// TwinCAT 3 PLC project AA_Planta_2324_MN
// ProgramVersion: 3.1.4024.0
// libraries:
//   Tc2_Standard, * (Beckhoff Automation GmbH)
//   Tc2_System, * (Beckhoff Automation GmbH)
//   Tc3_Module, * (Beckhoff Automation GmbH)
// project tree:
//   DUTs/ COLOR.TcDUT
//   DUTs/DefinicionCases/ CALMACENAMIENTO.TcDUT, CINTA.TcDUT, CPICKANDPLACE.TcDUT, CPOSITIONERLEFTBAR.TcDUT, CONDICIONESPARO.TcDUT, CRETIRADA.TcDUT, CTURNTABLE.TcDUT, STOPBLADE.TcDUT
//   DUTs/Objetos/ BeltConveyor.TcDUT, PickandPlace.TcDUT, PositioningLeftBar.TcDUT, Pusher.TcDUT, RollerConveyor.TcDUT, Selector.TcDUT, StrackerCraneRack.TcDUT, Turntable.TcDUT
//   GVLs/ GVL_General.TcGVL, GVL_ProcesoPallet.TcGVL, GVL_Sorting.TcGVL, GVL_StackBox.TcGVL, GVL_Almacen.TcGVL
//   / PlcTask.TcTTO
//   POUs/0_ControlEncendido/ PRG_FinDeCiclo.TcPOU, PRG_OnFabrica.TcPOU, PRG_SetaEmergencia.TcPOU, PRG_StopBladePyP.TcPOU
//   POUs/3_ProcesoPalet/ PRG_Cintas.TcPOU, PRG_Turntable.TcPOU
//   POUs/4_Almacen/ DINT_TO_COLOR.TcPOU, PRG_Almacen.TcPOU, PRG_PanelDeControl.TcPOU, PRG_RetiradaAlmacen.TcPOU
//   POUs/6_Contadores/ POU_Contadores.TcPOU
//   POUs/ MAIN.TcPOU
//   POUs/1_ProcesoEntrada/ FB_Pusher.TcPOU, PRG_ProcesoEntrada.TcPOU
//   POUs/2_ProcesoGuardado/ FB_Cinta.TcPOU, FB_PickAndPlace.TcPOU, FB_Positioner.TcPOU, FB_StopBlade.TcPOU, PRG_Parada.TcPOU, PRG_PickAndPlace.TcPOU, PRG_Positioner.TcPOU
// real-time tasks:
//   TASK PlcTask: cycle T#10ms, priority 20, ADS port 350
//   TASK PlcTask1: cycle T#10ms, priority 21, ADS port 351

CONFIGURATION AA_Planta_2324_MN
    RESOURCE PLC ON TwinCAT3
        TASK PlcTask(INTERVAL := T#10ms, PRIORITY := 21);
        PROGRAM MAIN WITH PlcTask : MAIN;
    END_RESOURCE
END_CONFIGURATION

// ---- DUTs/COLOR.TcDUT
{attribute 'strict'}
TYPE COLOR :
(
	AZUL := 2,
	VERDE := 5,
	METAL := 8,
	VACIO := 0
);
END_TYPE

// ---- DUTs/DefinicionCases/CALMACENAMIENTO.TcDUT
{attribute 'strict'}
TYPE CALMACENAMIENTO :
(
	CALMACEN_ESPERA,
	CALMACEN_MONTARPALLET,
	CALMACEN_BUSQUEDA,
	CALMACEN_GUARDADO,
	CALMACEN_LLENO,
	CALMACEN_ORIGEN
	
);
END_TYPE

// ---- DUTs/DefinicionCases/CINTA.TcDUT
{attribute 'strict'}
TYPE CINTA :
(
	CINTA_ACTIVADO,
	CINTA_REPOSO
);
END_TYPE

// ---- DUTs/DefinicionCases/CPICKANDPLACE.TcDUT
{attribute 'strict'}
TYPE CPICKANDPLACE :
(
	PICKANDPLACE_ESPERA,
	PICKANDPLACE_DETECCION,
	PICKANDPLACE_AGARRE,
	PICKANDPLACE_GIRO,
	PICKANDPLACE_COLOCACION,
	PICKANDPLACE_DESCENSO,
	PICKANDPLACE_LLENADO,
	PICKANDPLACE_ORIGEN
);
END_TYPE

// ---- DUTs/DefinicionCases/CPOSITIONERLEFTBAR.TcDUT
{attribute 'strict'}
TYPE CPOSITIONERLEFTBAR :
(
	CPOSITIONERLEFTBAR_ESPERA,
	CPOSITIONERLEFTBAR_AGARRE,
	CPOSITIONERLEFTBAR_PROCESADO,
	CPOSITIONERLEFTBAR_RESET,
	CPOSITIONERLEFTBAR_PASO
	
	
);
END_TYPE

// ---- DUTs/DefinicionCases/CONDICIONESPARO.TcDUT
{attribute 'strict'}
TYPE CONDICIONESPARO :
(
	CONDICIONESPARO_ESPERA,
	CONDICIONESPARO_SELECCION,
	CONDICIONESPARO_FINPROCESO,
	CONDICIONESPARO_ALMACEN,
	CONDICIONESPARO_SELECTOR,
	CONDICIONESPARO_GUARDADO,
	CONDICIONESPARO_CINTAINICIAL
);
END_TYPE

// ---- DUTs/DefinicionCases/CRETIRADA.TcDUT
{attribute 'strict'}
TYPE CRETIRADA :
(
	CRETIRADA_ESPERA,
	CRETIRADA_BUSQUEDA,
	CRETIRADA_RECOGIDA,
	CRETIRADA_TRANSPORTE,
	CRETIRADA_COLOCACION,
	CRETIRADA_PARTIDA
);
END_TYPE

// ---- DUTs/DefinicionCases/CTURNTABLE.TcDUT
{attribute 'strict'}
TYPE CTURNTABLE :
(
	CTURNTABLE_ESPERA,
	CTURNTABLE_FILTROPRIORIDAD,
	
	CTURNTABLE_ENTRADAVERDE,
	CTURNTABLE_CARGAVERDE,
	CTURNTABLE_DESCARGAVERDE,
	
	CTURNTABLE_ENTRADAAZUL,
	CTURNTABLE_CARGAAZUL,
	CTURNTABLE_DESCARGAAZUL,
	
	CTURNTABLE_ENTRADAMETAL,
	CTURNTABLE_CARGAMETAL,
	CTURNTABLE_DESCARGAMETAL,
	
	CTURNTABLE_COLOCACION,
	CTURNTABLE_SALIDA
);
END_TYPE

// ---- DUTs/DefinicionCases/STOPBLADE.TcDUT
{attribute 'strict'}
TYPE STOPBLADE :
(
	STOPBLADE_REPOSO,
	STOPBLADE_ACTIVADO
);
END_TYPE

// ---- DUTs/Objetos/BeltConveyor.TcDUT
{attribute 'OPC.UA.DA' := '1'}
TYPE BeltConveyor :
STRUCT
	
	(* Cintas comunes correspondientes al proceso de Sorting, ordenadas por aparición*)
	bSortingCintaInicial		: BOOL;
	bSortingCintaEntrada		: BOOL;
	bSortingCintaDistribucion	: BOOL;
	
	(* Cintas PARA PIEZAS AZULES, ordenadas por aparición*)
	bCintaAzul1 	: BOOL;
	bCintaAzul2		: BOOL;
	
	(* Cintas PARA PIEZAS VERDES, ordenadas por aparición*)
	bCintaVerde1 	: BOOL;
	bCintaVerde2	: BOOL;

	(* Cintas PARA PIEZAS METAL, ordenadas por aparición*)
	bCintaMetal1 	: BOOL;
	bCintaMetal2	: BOOL;
	
END_STRUCT
END_TYPE

// ---- DUTs/Objetos/PickandPlace.TcDUT
{attribute 'OPC.UA.DA' := '1'}
TYPE PickandPlace :
STRUCT
	
	(* Outputs del Pick and Place *)
 	bMovementZ 	: BOOL;
 	bMovementX 	: BOOL;
	bRotateCW 	: BOOL;
	bRotateCCW 	: BOOL;
	bGripperCW 	: BOOL;
	bGripperCCW : BOOL;
	bGrab 		: BOOL;
	
	(* Inputs del Pick and Place *)
	bMovingX 			: BOOL;
	bMovingZ 			: BOOL;
	bRotating 			: BOOL;
	bGripperRotating	: BOOL;
	bDetected 			: BOOL;

END_STRUCT
END_TYPE

// ---- DUTs/Objetos/PositioningLeftBar.TcDUT
{attribute 'OPC.UA.DA' := '1'}
TYPE PositioningLeftBar :
STRUCT
	
	(* Outputs del Positioning Left Bar *)
	bClamp : BOOL;
	bRaise : BOOL;
	
	(* Inputs del Positioning Left Bar *)
	bClamped : BOOL;
	bLimit	 : BOOL;
	
END_STRUCT
END_TYPE

// ---- DUTs/Objetos/Pusher.TcDUT
{attribute 'OPC.UA.DA' := '1'}
TYPE Pusher :
STRUCT
	Pusher: BOOL;
	PusherFrontLimit: BOOL;
	PusherBackLimit: BOOL;
END_STRUCT
END_TYPE

// ---- DUTs/Objetos/RollerConveyor.TcDUT
{attribute 'OPC.UA.DA' := '1'}
TYPE RollerConveyor :
STRUCT
	
	(* ROLL PARA PIEZAS AZULES, ordenadas por aparición*)
	bRollerAzul1 		 : BOOL;
	bCurvedRollerAzul1 	 : BOOL;
	
	(* ROLL PARA PIEZAS VERDES, ordenadas por aparición*)
	bRollerVerde1 		 : BOOL;
	
	(* ROLL PARA PIEZAS METAL, ordenadas por aparición*)
	bRollerMetal1 		 : BOOL;
	bCurvedRollerMetal1  : BOOL;
	
	(* ROLL ALMACEN, ordenadas por aparición*)
	bRollerAlmacen1		 : BOOL;
	bCurvedRollerAlmacen : BOOL;
	bRollerAlmacen2		 : BOOL;
	
	(* ROLLER SALIDA ALMACEN, ordenadas por aparición *)
	
	bRollerAlmacen3 : BOOL;
	bRollerAlmacen4 : BOOL;
	
END_STRUCT
END_TYPE

// ---- DUTs/Objetos/Selector.TcDUT
{attribute 'OPC.UA.DA' := '1'}
TYPE Selector :
STRUCT
	StateAzul : BOOL;
	StateMetal : BOOL;
END_STRUCT
END_TYPE

// ---- DUTs/Objetos/StrackerCraneRack.TcDUT
{attribute 'OPC.UA.DA' := '1'}
TYPE StrackerCraneRack :
STRUCT
	
	(* Outputs del Almacen *)
	TargetPosition: INT;
	Left:BOOL;
	Right:BOOL;
	Lift:BOOL;
	
	(* Inputs del Almacen *)
	MovingX:BOOL;
	MovingZ:BOOL;
	LeftLimit:BOOL;
	MiddleLimit:BOOL;
	RightLimit:BOOL;
	
END_STRUCT
END_TYPE

// ---- DUTs/Objetos/Turntable.TcDUT
{attribute 'OPC.UA.DA' := '1'}
TYPE Turntable :
STRUCT
	
	(* Outputs de la Turntable *)
	RollPositivo : BOOL;
	RollNegativo : BOOL;
	Turn		 : BOOL;
	
	(* Inputs de la Turntable *)
	FrontLimit	 : BOOL;
	BackLimit	 : BOOL;
	Limit0		 : BOOL;
	Limit90		 : BOOL;
	
END_STRUCT
END_TYPE

// ---- GVLs/GVL_General.TcGVL
{attribute 'qualified_only'}
VAR_GLOBAL
	{attribute 'OPC.UA.DA' := '1'}
	bMarcha : BOOL;
	{attribute 'OPC.UA.DA' := '1'}
	bParo : BOOL;
	{attribute 'OPC.UA.DA' := '1'}
	bSetaEmergencia : BOOL;
	
	{attribute 'OPC.UA.DA.StructuredType' := '1'}
	sBeltConveyor: BeltConveyor;
	
	{attribute 'OPC.UA.DA' := '1'}
	bStopBlade1 : BOOL;	
	
END_VAR

// ---- GVLs/GVL_ProcesoPallet.TcGVL
{attribute 'qualified_only'}
VAR_GLOBAL	
	
	{attribute 'OPC.UA.DA.StructuredType' := '1'}
	sTurnTable: Turntable;
	{attribute 'OPC.UA.DA.StructuredType' := '1'}
	sRollerConveyor: RollerConveyor;
	
	{attribute 'OPC.UA.DA' := '1'}
	bDiffuseSensorPaletA	:BOOL;
	{attribute 'OPC.UA.DA' := '1'}
	bDiffuseSensorPaletV	:BOOL;
	{attribute 'OPC.UA.DA' := '1'}
	bDiffuseSensorPaletM	:BOOL;
	{attribute 'OPC.UA.DA' := '1'}	
	bDiffuseSensorSalida		:BOOL;
	
	{attribute 'OPC.UA.DA' := '1'}
	iLightArrayEmitterA		:BOOL;
	{attribute 'OPC.UA.DA' := '1'}
	iLightArrayEmitterV		:BOOL;
	{attribute 'OPC.UA.DA' := '1'}
	iLightArrayEmitterM		:BOOL; 
	
END_VAR

// ---- GVLs/GVL_Sorting.TcGVL
{attribute 'qualified_only'}
VAR_GLOBAL

	(* Variables correspondientes al proceso de sorting de las piezas AZULES *)
	{attribute 'OPC.UA.DA' := '1'}
	bVisionSensorA	: BOOL;
	{attribute 'OPC.UA.DA.StructuredType' := '1'}
	sPusherA: Pusher;
	{attribute 'OPC.UA.DA' := '1'}
	bDiffuseSensorA: BOOL;
	
	(* Variables correspondientes al proceso de sorting de las piezas VERDES *)
	{attribute 'OPC.UA.DA.StructuredType' := '1'}
	sPusherV: Pusher;
	{attribute 'OPC.UA.DA' := '1'}
	bVisionSensorV	: BOOL;	
	{attribute 'OPC.UA.DA' := '1'}
	bDiffuseSensorV: BOOL;
	
	(* Variables correspondientes al proceso de sorting de las piezas METÁLICAS *)
	{attribute 'OPC.UA.DA.StructuredType' := '1'}
	sPusherM: Pusher;
	{attribute 'OPC.UA.DA' := '1'}
	bVisionSensorM	: BOOL;
	{attribute 'OPC.UA.DA' := '1'}
	bDiffuseSensorM: BOOL;
	
END_VAR

// ---- GVLs/GVL_StackBox.TcGVL
{attribute 'qualified_only'}
VAR_GLOBAL
	
	(* Variables correspondientes a la Línea Azul*)
	
	{attribute 'OPC.UA.DA.StructuredType' := '1'}
	sPickAndPlaceA	: PickAndPlace;
	{attribute 'OPC.UA.DA.StructuredType' := '1'}
	sPosLeftBarA	: PositioningLeftBar;
	{attribute 'OPC.UA.DA' := '1'}
	bStopBladeA1: BOOL;
	{attribute 'OPC.UA.DA' := '1'}
	bStopBladeA2: BOOL := TRUE;
	
	{attribute 'OPC.UA.DA' := '1'}
	bRReflectiveSensorA1 	: BOOL	:= TRUE;
	{attribute 'OPC.UA.DA' := '1'}
	bRReflectiveSensorA2 	: BOOL	:= TRUE;
	{attribute 'OPC.UA.DA' := '1'}
	bRReflectiveSensorA3	: BOOL	:= TRUE;
	{attribute 'OPC.UA.DA' := '1'}
	bDiffuseSensorPyPA		: BOOL	:= FALSE;
	

	
	(* Variables correspondientes a la Línea Verde*)
	
	{attribute 'OPC.UA.DA.StructuredType' := '1'}
	sPickAndPlaceV	: PickAndPlace;
	{attribute 'OPC.UA.DA.StructuredType' := '1'}
	sPosLeftBarV	: PositioningLeftBar;
	{attribute 'OPC.UA.DA' := '1'}
	bStopBladeV1: BOOL;
	{attribute 'OPC.UA.DA' := '1'}
	bStopBladeV2: BOOL := TRUE;
	
	
	{attribute 'OPC.UA.DA' := '1'}
	bRReflectiveSensorV1 : BOOL		:= TRUE;
	{attribute 'OPC.UA.DA' := '1'}
	bRReflectiveSensorV2 : BOOL		:= TRUE;
	{attribute 'OPC.UA.DA' := '1'}	
	bRReflectiveSensorV3 : BOOL		:= TRUE;
	{attribute 'OPC.UA.DA' := '1'}	
	bDiffuseSensorPyPV	 : BOOL		:= FALSE;
	
	
	
	(* Variables correspondientes a la Línea Metal*)
	
	{attribute 'OPC.UA.DA.StructuredType' := '1'}
	sPickAndPlaceM	: PickAndPlace;
	{attribute 'OPC.UA.DA.StructuredType' := '1'}
	sPosLeftBarM	: PositioningLeftBar;
	{attribute 'OPC.UA.DA' := '1'}
	bStopBladeM1: BOOL;
	{attribute 'OPC.UA.DA' := '1'}
	bStopBladeM2: BOOL := TRUE;
	
	{attribute 'OPC.UA.DA' := '1'}
	bRReflectiveSensorM1 : BOOL		:= TRUE;
	{attribute 'OPC.UA.DA' := '1'}
	bRReflectiveSensorM2 : BOOL		:= TRUE;
	{attribute 'OPC.UA.DA' := '1'}
	bRReflectiveSensorM3 : BOOL		:= TRUE;
	{attribute 'OPC.UA.DA' := '1'}
	bDiffuseSensorPyPM	 : BOOL		:= FALSE;

END_VAR

// ---- GVLs/GVL_Almacen.TcGVL
{attribute 'qualified_only'}
VAR_GLOBAL
	
	(* Sensores y actuadores asociados al ciclo del Almacén*)
	
	{attribute 'OPC.UA.DA.StructuredType' := '1'}
	sStackCraneRack: StrackerCraneRack;
	
	{attribute 'OPC.UA.DA' := '1'}
	bDifusseSensorAlmacen:BOOL;
	{attribute 'OPC.UA.DA' := '1'}
	iVisionSensorAlmacen: DINT;
	{attribute 'OPC.UA.DA' := '1'}
	bRRflexSensorAlmacen:BOOL;
	
	{attribute 'OPC.UA.DA' := '1'}
	bLoadingConveyor:BOOL;
	
	(* Almacenamiento de datos de las diferentes posiciones (no es necesario que sea una GVL) *)
	aAlmacen: ARRAY[1..54] OF COLOR  :=[54(0)];
	

	(* Memoria del color solicitado (no es necesario que sea una GVL) *)
	iSolicitudColor : INT;
	
	(* Botones de activación, paro y seta y elementos asociados al panel del Almacén *)
	
	{attribute 'OPC.UA.DA' := '1'}
	Sacar: BOOL;
	{attribute 'OPC.UA.DA' := '1'}
	bReset: BOOL;
	{attribute 'OPC.UA.DA' := '1'}
	bSetaEmergencia: BOOL;
	
	{attribute 'OPC.UA.DA.StructuredType' := '1'}
	sSelector : Selector;
	
	{attribute 'OPC.UA.DA' := '1'}
	iDisplay : INT;
	{attribute 'OPC.UA.DA' := '1'}
	LedAzul: BOOL;
	{attribute 'OPC.UA.DA' := '1'}
	LedVerde: BOOL;
	{attribute 'OPC.UA.DA' := '1'}
	LedMetal: BOOL;
	
END_VAR

// ---- POUs/MAIN.TcPOU
PROGRAM MAIN
VAR
	bON: BOOL; 
END_VAR

(*
  	  ESCOLA POLITÉCNICA DE ENXEÑARÍA DE FERROL			
			  UNIVERSIDADE DA CORUÑA 						
			
Máster Universitario en Informática Industrial y Robótica   
  	Automatización Avanzada - Curso 2023-2024			

					Profesorado: 						
 	Antonio J. Díaz Longueira - Míriam Timiraos Díaz 		

 		    	Código realizado por:
	Marta María Álvarez Crespo - Noelia Pita López  		
*)



(* PRGs siempre activos, necesarios para el correcto control de la fábrica *)
PRG_StopBladePyP();
POU_Contadores();


(* Cuando se pulsa el botón verde, se activa la fábrica y solo se detendrá en caso de que se pulse el botón de paro o la seta de emergencia.
En el caso del botón de paro, desactivará el valor de bON de forma que se llame a un POU diferente a los llamados en este MAIN, donde el proceso
se detiene progresivamente *)

IF GVL_General.bMarcha THEN
	bON := TRUE;
END_IF

IF NOT GVL_General.bParo THEN
	bON := FALSE;
END_IF

IF NOT bON THEN
	PRG_FinDeCiclo();
END_IF


IF bON AND GVL_General.bSetaEmergencia THEN
	
	PRG_OnFabrica();
	PRG_ProcesoEntrada();
	PRG_PickAndPlace();
	PRG_Positioner();
	PRG_Parada();
	PRG_Turntable();
	PRG_Almacen();
	PRG_Cintas();
	PRG_PaneldeControl();
	
	IF GVL_Almacen.bSetaEmergencia THEN
		PRG_RetiradaAlmacen();
	END_IF
	
END_IF

IF NOT GVL_General.bSetaEmergencia THEN
	PRG_SetaEmergencia();
END_IF





























































(*
		♡ 
    /\_____/\
   /  o   o  \						
  ( ==  ^  == )		
   )         (		   __     miau
 (             )______/  |		miau 
(__(__)___(__)__)_______/	 

*)

END_PROGRAM

// ---- POUs/0_ControlEncendido/PRG_StopBladePyP.TcPOU
PROGRAM PRG_StopBladePyP
VAR
END_VAR

GVL_StackBox.bStopBladeA2 := TRUE;
GVL_StackBox.bStopBladeV2 := TRUE;
GVL_StackBox.bStopBladeM2 := TRUE;

END_PROGRAM

// ---- POUs/6_Contadores/POU_Contadores.TcPOU
PROGRAM POU_Contadores
VAR
	iCintaProcesando : INT := 0;
	iStackBoxProcesando: INT := 0;
	iCajaProcesando : INT := 0;
	bGuardandoCaja: BOOL := 0;
	iProcesandoCintas: INT := 0;
	
	reDifSensorSorting: R_TRIG;
	feRRefSensorSortingA: F_TRIG;
	feRRefSensorSortingV: F_TRIG;
	reDifSensorSortingM: F_TRIG;
	fTrigRRefSensorAlmacen: F_TRIG;
	tFTrigEmitterA: F_TRIG;
	tFTrigEmitterV: F_TRIG;
	tFTrigEmitterM: F_TRIG;
	tFTrigDiffuseSensor : F_TRIG;
	
	fFtrigRobotSeMueveA : F_TRIG;
	fFtrigRobotSeMueveV : F_TRIG;
	fFtrigRobotSeMueveM : F_TRIG;
END_VAR

reDifSensorSorting(CLK:= GVL_Sorting.bDiffuseSensorA);
feRRefSensorSortingA(CLK:= GVL_StackBox.bRReflectiveSensorA1);
feRRefSensorSortingV (CLK:= GVL_StackBox.bRReflectiveSensorV1); 
reDifSensorSortingM (CLK:= GVL_Sorting.bDiffuseSensorM);
tFTrigDiffuseSensor(CLK:= GVL_ProcesoPallet.bDiffuseSensorSalida);
fTrigRRefSensorAlmacen(CLK:= GVL_Almacen.bRRflexSensorAlmacen);
tFTrigEmitterA(CLK:= GVL_ProcesoPallet.iLightArrayEmitterA);
tFTrigEmitterV(CLK:= GVL_ProcesoPallet.iLightArrayEmitterV);
tFTrigEmitterM(CLK:= GVL_ProcesoPallet.iLightArrayEmitterM);

fFtrigRobotSeMueveA(CLK:= PRG_PickAndPlace.RobotSeMueveA);
fFtrigRobotSeMueveV(CLK:= PRG_PickAndPlace.RobotSeMueveV);
fFtrigRobotSeMueveM(CLK:= PRG_PickAndPlace.RobotSeMueveM);

// SECCION 1 
(* Sumamos 1 al contador si se comienza a procesar una pieza y se resta 1 cuando se termina de procesar *)

IF reDifSensorSorting.Q THEN
	iCintaProcesando := iCintaProcesando + 1;
END_IF

IF feRRefSensorSortingA.Q THEN
	iCintaProcesando := iCintaProcesando - 1;
END_IF

IF feRRefSensorSortingV.Q THEN
	iCintaProcesando := iCintaProcesando - 1;
END_IF

IF reDifSensorSortingM.Q THEN
	iCintaProcesando := iCintaProcesando - 1;
END_IF


// SECCION 2 
(* Sumamos 1 al contador si se comienza a procesar una pieza y se resta 1 cuando se termina de procesar *)

IF feRRefSensorSortingA.Q THEN
	iStackBoxProcesando := iStackBoxProcesando + 1;
END_IF

IF feRRefSensorSortingV.Q THEN
	iStackBoxProcesando := iStackBoxProcesando + 1;
END_IF

IF reDifSensorSortingM.Q THEN
	iStackBoxProcesando := iStackBoxProcesando + 1;
END_IF


IF fFtrigRobotSeMueveA.Q THEN
	iStackBoxProcesando := iStackBoxProcesando - 1;
END_IF

IF fFtrigRobotSeMueveV.Q THEN
	iStackBoxProcesando := iStackBoxProcesando - 1;
END_IF

IF fFtrigRobotSeMueveM.Q THEN
	iStackBoxProcesando := iStackBoxProcesando - 1;
END_IF

// SECCION 3 
(* Sumamos 1 al contador si se comienza a procesar una pieza y se resta 1 cuando se termina de procesar *)

IF tFTrigEmitterV.Q THEN
	iCajaProcesando := iCajaProcesando + 1;
END_IF

IF tFTrigEmitterA.Q THEN
	iCajaProcesando := iCajaProcesando + 1;
END_IF

IF tFTrigEmitterM.Q THEN
	iCajaProcesando := iCajaProcesando + 1;
END_IF

IF tFTrigDiffuseSensor.Q THEN
	iCajaProcesando := iCajaProcesando - 1;
END_IF


// SECCION 4
(* Sumamos 1 al contador si se comienza a procesar una pieza a través de los roller conveyor y restamos cuando termina de procesar *)

IF tFTrigDiffuseSensor.Q THEN
	iProcesandoCintas := iProcesandoCintas + 1;
END_IF

IF fTrigRRefSensorAlmacen.Q THEN
	iProcesandoCintas := iProcesandoCintas - 1;
END_IF


// SECCION 5 
(* Sumamos 1 al contador si se comienza a procesar una pieza y se resta 1 cuando se termina de procesar *)

IF PRG_Almacen.ALMACEN > 1 THEN
	bGuardandoCaja := TRUE;
END_IF

IF PRG_Almacen.ALMACEN < 2 THEN
	bGuardandoCaja := FALSE;
END_IF

END_PROGRAM

// ---- POUs/2_ProcesoGuardado/PRG_PickAndPlace.TcPOU
PROGRAM PRG_PickAndPlace
VAR
(* =============================================================================================== *)
(*                                CONTROL DE LOS PICK-AND-PLACE                                    *)
(* =============================================================================================== *)

// PIEZAS AZULES	
	PickAndPlaceA: FB_PickAndPlace;
	
	RobotSeMueveA: BOOL;
	iContadorPyPA: INT;
	CajaLlenaA: BOOL;
	
// PIEZAS VERDES
	PickAndPlaceV: FB_PickAndPlace;
	
	RobotSeMueveV: BOOL;
	iContadorPyPV: INT;
	CajaLlenaV: BOOL;
	
// PIEZAS METAL
	PickAndPlaceM: FB_PickAndPlace;
	
	RobotSeMueveM: BOOL;
	iContadorPyPM: INT;
	CajaLlenaM: BOOL;
END_VAR

(* El Pick-and-Place se encarga de llevar el material a su correspondiente caja. Para ello, se plantea el 
uso de un CASE para controlar la posición del brazo, dividiendo su proceso por etapas *)

// PIEZAS AZULES
PickAndPlaceA(
	MOVIENDOZ:= GVL_StackBox.sPickAndPlaceA.bMovingZ, MOVIENDOX:= GVL_StackBox.sPickAndPlaceA.bMovingX, 
	ROTANDO:= GVL_StackBox.sPickAndPlaceA.bRotating, DETECTADO:= GVL_StackBox.sPickAndPlaceA.bDetected, 
	SENSOR:= GVL_StackBox.bDiffuseSensorPyPA, RESET := PRG_Turntable.tRTrigEmitterA.Q, ROBOTSEMUEVE=> RobotSeMueveA, 
	MOVERZ=> GVL_StackBox.sPickAndPlaceA.bMovementZ, MOVERX=> GVL_StackBox.sPickAndPlaceA.bMovementX, 
	ROTARCCW=> GVL_StackBox.sPickAndPlaceA.bRotateCCW, ROTARCW=> GVL_StackBox.sPickAndPlaceA.bRotateCW, 
	AGARRAR=> GVL_StackBox.sPickAndPlaceA.bGrab, CAJALLENA => CajaLlenaA);
		

// PIEZAS VERDES
PickAndPlaceV(
	MOVIENDOZ:= GVL_StackBox.sPickAndPlaceV.bMovingZ, MOVIENDOX:= GVL_StackBox.sPickAndPlaceV.bMovingX, 
	ROTANDO:= GVL_StackBox.sPickAndPlaceV.bRotating, DETECTADO:= GVL_StackBox.sPickAndPlaceV.bDetected, 
	SENSOR:= GVL_StackBox.bDiffuseSensorPyPV, RESET := PRG_Turntable.tRTrigEmitterV.Q, ROBOTSEMUEVE=> RobotSeMueveV, 
	MOVERZ=> GVL_StackBox.sPickAndPlaceV.bMovementZ, MOVERX=> GVL_StackBox.sPickAndPlaceV.bMovementX, 
	ROTARCCW=> GVL_StackBox.sPickAndPlaceV.bRotateCCW, ROTARCW=> GVL_StackBox.sPickAndPlaceV.bRotateCW, 
	AGARRAR=> GVL_StackBox.sPickAndPlaceV.bGrab, CAJALLENA => CajaLlenaV);
		
// PIEZAS METAL
PickAndPlaceM(
	MOVIENDOZ:= GVL_StackBox.sPickAndPlaceM.bMovingZ, MOVIENDOX:= GVL_StackBox.sPickAndPlaceM.bMovingX, 
	ROTANDO:= GVL_StackBox.sPickAndPlaceM.bRotating, DETECTADO:= GVL_StackBox.sPickAndPlaceM.bDetected, 
	SENSOR:= GVL_StackBox.bDiffuseSensorPyPM, RESET := PRG_Turntable.tRTrigEmitterM.Q, ROBOTSEMUEVE=> RobotSeMueveM, 
	MOVERZ=> GVL_StackBox.sPickAndPlaceM.bMovementZ, MOVERX=> GVL_StackBox.sPickAndPlaceM.bMovementX, 
	ROTARCCW=> GVL_StackBox.sPickAndPlaceM.bRotateCCW, ROTARCW=> GVL_StackBox.sPickAndPlaceM.bRotateCW, 
	AGARRAR=> GVL_StackBox.sPickAndPlaceM.bGrab, CAJALLENA => CajaLlenaM);

END_PROGRAM

// ---- POUs/2_ProcesoGuardado/FB_PickAndPlace.TcPOU
FUNCTION_BLOCK FB_PickAndPlace
VAR_INPUT
	
	MOVIENDOZ: BOOL;
	MOVIENDOX: BOOL;
	ROTANDO: BOOL;
	DETECTADO: BOOL;
	SENSOR: BOOL;
	
	RESET: BOOL;
	
END_VAR

VAR_OUTPUT
	
	ROBOTSEMUEVE: BOOL;
	
	MOVERZ: BOOL;
	MOVERX: BOOL;
	ROTARCCW: BOOL;
	ROTARCW: BOOL;
	AGARRAR: BOOL;
	CAJALLENA: BOOL;
	
END_VAR

VAR
	CONTADOR: CTU;	
	CPICKANDPLACE: CPICKANDPLACE;
	bFTrigMovingX: F_TRIG;
	bFTrigMovingZ: F_TRIG;
	bFTrigRotating: F_TRIG;
	bFTrigDetected: F_TRIG;
	bRTrigDetected: R_TRIG;
	bRTrigDiffSensorPyP: R_TRIG;		
	bConterTrigger: F_TRIG;
	tRecogidaBrazo: TON;
END_VAR

bFTrigMovingZ(CLK:= MOVIENDOZ);
bFTrigMovingX(CLK:= MOVIENDOX);
bFTrigRotating(CLK:= ROTANDO);
bRTrigDetected(CLK:= DETECTADO);
bFTrigDetected(CLK:= DETECTADO);
bRTrigDiffSensorPyP(CLK:= SENSOR);
bConterTrigger(CLK:= ROTARCW);
tRecogidaBrazo(IN:= NOT MOVERZ, PT:= T#1S);

CONTADOR(CU:= bConterTrigger.Q, RESET:=RESET, PV:= 3, Q=> CAJALLENA);

CASE CPICKANDPLACE OF
	
	PICKANDPLACE_ESPERA:
	(* La maquina esta esperando a que sea su turno para funcionar *)
		
		IF bRTrigDiffSensorPyP.Q THEN
			CPICKANDPLACE := PICKANDPLACE_DETECCION;
		END_IF

	
	PICKANDPLACE_DETECCION:
	(* Cuando se detecta un LID posicionado, se baja el brazo hasta su detección *)
		
		ROBOTSEMUEVE := TRUE;
		IF NOT CONTADOR.Q THEN
			MOVERZ := TRUE;
			CPICKANDPLACE := PICKANDPLACE_AGARRE;
		END_IF
		
	
	PICKANDPLACE_AGARRE: 
	(* Se agarra el LID detectado una vez detenido el movimiento de Z y se sube el brazo de nuevo *)
	
		IF bRTrigDetected.Q THEN
			AGARRAR := TRUE;
			MOVERZ := FALSE;
			CPICKANDPLACE := PICKANDPLACE_GIRO;	
		END_IF
		
		
	PICKANDPLACE_GIRO:
	(* Se comprueba que el brazo está bien posicionado y se rota hacia la sección de llenado de cajas *)
		
		IF bFTrigMovingZ.Q THEN
			ROTARCCW := TRUE;
		END_IF
		
		IF bFTrigRotating.Q THEN
			ROTARCCW := FALSE;
			CPICKANDPLACE := PICKANDPLACE_COLOCACION;	
		END_IF
	
	
	PICKANDPLACE_COLOCACION:
	(* Cuando se posiciona sobre la zona de llenado de la caja, se estira para achinar dentro *)
	
		MOVERX := TRUE;
		
		IF bFTrigMovingX.Q THEN
			CPICKANDPLACE := PICKANDPLACE_DESCENSO;
		END_IF
	
	
	PICKANDPLACE_DESCENSO: 
	(* Cuando termina de estirarse, vuelve a bajar el brazo para depositar el LID en la caja *)
	
		MOVERZ:= TRUE;		
		IF bFTrigMovingZ.Q THEN
			CPICKANDPLACE := PICKANDPLACE_LLENADO;
		END_IF
	
	
	PICKANDPLACE_LLENADO:
	(* Cuando se termina de mover en Z, deposita el LID en la caja abriendo el Gripper y sube a su posicion 0 *)
	
		AGARRAR := FALSE;	
		MOVERZ := FALSE;
		
		IF tRecogidaBrazo.Q THEN
			MOVERX := FALSE;	
		END_IF	
		
		IF bFTrigMovingX.Q THEN
			CPICKANDPLACE := PICKANDPLACE_ORIGEN;	
		END_IF	
	
		
	PICKANDPLACE_ORIGEN:
	(* El brazo vuelve a su posición inicial e inicia un nuevo ciclo *)

		ROTARCW := TRUE;	
		
		IF bFTrigRotating.Q THEN 
			ROTARCW := FALSE;
			ROBOTSEMUEVE := FALSE;
			CPICKANDPLACE := PICKANDPLACE_ESPERA;
		END_IF
		
END_CASE

END_FUNCTION_BLOCK

// ---- POUs/3_ProcesoPalet/PRG_Turntable.TcPOU
PROGRAM PRG_Turntable
VAR
	// Asignación de valores del CASE
	Turntable : CTURNTABLE;
	
	// FB asociados a cambios de flanco, timers...
	tFTrigDiffuseSensor	: F_TRIG;
	tFTrigEmitterA		: F_TRIG;
	tFTrigEmitterV		: F_TRIG;
	tFTrigEmitterM		: F_TRIG;
	tRTrigEmitterA		: R_TRIG;
	tRTrigEmitterV		: R_TRIG;
	tRTrigEmitterM		: R_TRIG;
	tRtrigCajaLlenaA	: R_TRIG;
	tRtrigCajaLlenaV	: R_TRIG;
	tRtrigCajaLlenaM	: R_TRIG;
	
	// Declaración de memorias para determinar qué camino se activará
	bMemoriaAzul: BOOL;
	bMemoriaVerde: BOOL;
	bMemoriaMetal: BOOL;
	
END_VAR

tFTrigDiffuseSensor(CLK:= GVL_ProcesoPallet.bDiffuseSensorSalida);
tFTrigEmitterA(CLK:= GVL_ProcesoPallet.iLightArrayEmitterA);
tFTrigEmitterV(CLK:= GVL_ProcesoPallet.iLightArrayEmitterV);
tFTrigEmitterM(CLK:= GVL_ProcesoPallet.iLightArrayEmitterM);
tRTrigEmitterA(CLK:= GVL_ProcesoPallet.iLightArrayEmitterA);
tRTrigEmitterV(CLK:= GVL_ProcesoPallet.iLightArrayEmitterV);
tRTrigEmitterM(CLK:= GVL_ProcesoPallet.iLightArrayEmitterM);
tRtrigCajaLlenaA(CLK:= PRG_PickAndPlace.CajaLlenaA);
tRtrigCajaLlenaV(CLK:= PRG_PickAndPlace.CajaLlenaV);
tRtrigCajaLlenaM(CLK:= PRG_PickAndPlace.CajaLlenaM);


// Activación de los Roller que envían las cajas al almacén
GVL_ProcesoPallet.sRollerConveyor.bCurvedRollerAlmacen := TRUE;
GVL_ProcesoPallet.sRollerConveyor.bRollerAlmacen1 := TRUE;
GVL_ProcesoPallet.sRollerConveyor.bRollerAlmacen2 := TRUE;


(* Para el procesado de esta estación, se generan una serie de variables que permiten que la máquina de estados propuesta, solo pueda
elegir un único camino. De esta manera, se parte de un estado inicial de reposo y, en cuanto las cajas alcanzan su valor máximo de llenado
a través del contador implementado en los PickAndPlace, la máquina saltará al estado correspondiente y procesará una de las líneas únicamente *)

IF tRtrigCajaLlenaA.Q THEN
	bMemoriaAzul := TRUE;
END_IF

IF tRtrigCajaLlenaV.Q THEN
	bMemoriaVerde := TRUE;
END_IF

IF tRtrigCajaLlenaM.Q THEN
	bMemoriaMetal := TRUE;
END_IF


CASE Turntable OF
	
	CTURNTABLE_ESPERA:
	(* Proceso espera *)
	
		IF bMemoriaAzul THEN
			TURNTABLE := CTURNTABLE_CARGAAZUL;
		END_IF
		
		
		IF bMemoriaVerde THEN
			TURNTABLE := CTURNTABLE_CARGAVERDE;
		END_IF
		
		
		IF bMemoriaMetal THEN
			TURNTABLE := CTURNTABLE_CARGAMETAL;
		END_IF
	
	CTURNTABLE_CARGAAZUL:
	(* Proceso de carga para la caja azul *)
	
		IF GVL_ProcesoPallet.bDiffuseSensorPaletA THEN
			GVL_ProcesoPallet.sRollerConveyor.bRollerAzul1 := FALSE;
			GVL_ProcesoPallet.sRollerConveyor.bCurvedRollerAzul1 := FALSE;
		ELSE
			GVL_ProcesoPallet.sRollerConveyor.bRollerAzul1 := TRUE;
			GVL_ProcesoPallet.sRollerConveyor.bCurvedRollerAzul1 := TRUE;
		END_IF
		
		GVL_ProcesoPallet.sTurnTable.Turn := TRUE;
		GVL_ProcesoPallet.sTurnTable.RollPositivo := TRUE;
		
		IF GVL_ProcesoPallet.sTurnTable.Limit90 THEN
			TURNTABLE := CTURNTABLE_DESCARGAAZUL;
		END_IF	
	
	
	CTURNTABLE_DESCARGAAZUL:
	(* Proceso de descarga para la caja azul *)
	
		GVL_ProcesoPallet.sRollerConveyor.bCurvedRollerAzul1 := TRUE;
		IF GVL_ProcesoPallet.sTurnTable.FrontLimit THEN
			GVL_ProcesoPallet.sTurnTable.RollPositivo := FALSE;
			GVL_ProcesoPallet.sTurnTable.Turn := FALSE;
		END_IF
		
		IF GVL_ProcesoPallet.sTurnTable.Limit0 THEN
			GVL_ProcesoPallet.sTurnTable.RollPositivo := TRUE;
			bMemoriaAzul := FALSE;
			TURNTABLE := CTURNTABLE_SALIDA;
		END_IF
		
	
	CTURNTABLE_CARGAVERDE:
	(* Proceso de carga para la caja verde *)
	
		IF GVL_ProcesoPallet.bDiffuseSensorPaletV THEN
			GVL_ProcesoPallet.sRollerConveyor.bRollerVerde1 := FALSE;
		ELSE
			GVL_ProcesoPallet.sRollerConveyor.bRollerVerde1 := TRUE;
		END_IF
		
		GVL_ProcesoPallet.sTurnTable.Turn := FALSE;
		
		IF GVL_ProcesoPallet.sTurnTable.Limit0 THEN
			GVL_ProcesoPallet.sRollerConveyor.bRollerVerde1 := TRUE;
			GVL_ProcesoPallet.sTurnTable.RollPositivo := TRUE;
			bMemoriaVerde := FALSE;
			TURNTABLE := CTURNTABLE_SALIDA;
		END_IF
	
	
	CTURNTABLE_CARGAMETAL:
	(* Proceso de carga para la caja azul *)
	
		IF GVL_ProcesoPallet.bDiffuseSensorPaletM THEN
			GVL_ProcesoPallet.sRollerConveyor.bRollerMetal1 := FALSE;
			GVL_ProcesoPallet.sRollerConveyor.bCurvedRollerMetal1 := FALSE;
		ELSE
			GVL_ProcesoPallet.sRollerConveyor.bRollerMetal1 := TRUE;
			GVL_ProcesoPallet.sRollerConveyor.bCurvedRollerMetal1 := TRUE;
		END_IF
		
		GVL_ProcesoPallet.sTurnTable.Turn := TRUE;
		GVL_ProcesoPallet.sTurnTable.RollNegativo := TRUE;
		
		IF GVL_ProcesoPallet.sTurnTable.Limit90 THEN
			TURNTABLE := CTURNTABLE_DESCARGAMETAL;
		END_IF	
		
	
	CTURNTABLE_DESCARGAMETAL:
	(* Proceso de descarga para la caja azul *)
	
		GVL_ProcesoPallet.sRollerConveyor.bCurvedRollerMetal1 := TRUE;
		IF GVL_ProcesoPallet.sTurnTable.BackLimit THEN
			GVL_ProcesoPallet.sTurnTable.RollNegativo := FALSE;
			GVL_ProcesoPallet.sTurnTable.Turn := FALSE;
		END_IF
		
		IF GVL_ProcesoPallet.sTurnTable.Limit0 THEN
			GVL_ProcesoPallet.sTurnTable.RollPositivo := TRUE;
			bMemoriaMetal := FALSE;
			TURNTABLE := CTURNTABLE_SALIDA;
		END_IF
	
	
	CTURNTABLE_SALIDA:
	(* Proceso de detección para determinar si la caja ya salió de la zona de acción de la mesa 
	   y poder comenzar el procesamiento de otras cajas *)
	   
		IF tFTrigDiffuseSensor.Q THEN
			TURNTABLE := CTURNTABLE_ESPERA;
			GVL_ProcesoPallet.sTurnTable.RollPositivo := FALSE;
		END_IF
	
END_CASE

END_PROGRAM

// ---- POUs/4_Almacen/PRG_Almacen.TcPOU
PROGRAM PRG_Almacen
VAR
	
	// Variables de control para conocer el estado de la máquina y permitir su coordinación con el proceso de retirada del almacén
	bEstoyLleno: BOOL;
	bAlmacenOcupado : BOOL;
	bAlmacenGuardando: BOOL;
	
	// Variables para almacenar la posición de almacenamiento y para el control del FOR
	iPosicion : INT;
	i: INT := 1;
	
	// VALORES DEL CASE
	ALMACEN: CALMACENAMIENTO;
	
	// Almacenamiento del tipo de caja almacenado para su escritura en el array
	LECTURA: COLOR;
	
	// Function Blocks de cambios de flanco, timers...
	fTrigRRefSensorAlmacen	: F_TRIG;
	fTrigLift				: F_TRIG;
	fTrigMovingX			: F_TRIG;
	tTimerRack 				: TON;

END_VAR

VAR_INPUT
	
	// Almacenamiento de la cantidad de cajas de cada color
	iCantidadAzul : INT;
	iCantidadVerde : INT;
	iCantidadMetal : INT;
	
END_VAR

fTrigRRefSensorAlmacen(CLK:= GVL_Almacen.bRRflexSensorAlmacen);
fTrigLift(CLK:= GVL_Almacen.sStackCraneRack.MovingZ);
fTrigMovingX(CLK:= GVL_Almacen.sStackCraneRack.MovingX);
tTimerRack(IN:=GVL_Almacen.sStackCraneRack.MiddleLimit, PT:=T#1S);

(* Este PRG se encarga de gestionar el almacenamiento en las estanterías. Para ello, comprueba si hay una caja lista para ser almacenada a través del resultado 
devuelto por el VisualSensor y la comprobación de que el almacén no esté realizando otras tareas en ese momento *)

IF GVL_Almacen.iVisionSensorAlmacen > 0 AND (bAlmacenOcupado OR PRG_RetiradaAlmacen.AlmacenSacando)THEN
	GVL_ProcesoPallet.sRollerConveyor.bRollerAlmacen2 := FALSE;
ELSE
	GVL_ProcesoPallet.sRollerConveyor.bRollerAlmacen2 := TRUE;
END_IF


(* Para ello, se define un CASE que realiza las diferentes lecturas y actuaciones necesarias para el correcto almacenamiento de las cajas *)

CASE ALMACEN OF
	
	CALMACEN_ESPERA:
	(* Colocamos el almacen en posición de espera *)
		
		IF NOT PRG_RetiradaAlmacen.AlmacenSacando THEN
			GVL_Almacen.sStackCraneRack.TargetPosition := 55;
			GVL_Almacen.bLoadingConveyor := FALSE;
			
			IF NOT GVL_Almacen.sStackCraneRack.MovingX AND NOT GVL_Almacen.sStackCraneRack.MovingZ AND tTimerRack.Q THEN
				GVL_Almacen.sStackCraneRack.Right := TRUE;
				GVL_Almacen.sStackCraneRack.Lift  := FALSE;
			END_IF
			
			IF GVL_Almacen.sStackCraneRack.RightLimit THEN
				bAlmacenGuardando := FALSE;
				bAlmacenOcupado := FALSE;
				ALMACEN := CALMACEN_MONTARPALLET;
			END_IF
		END_IF
	
	CALMACEN_MONTARPALLET:
	(* Esperamos a montar el palet en el almacén *)
	
		IF NOT PRG_RetiradaAlmacen.AlmacenSacando THEN	
			IF GVL_Almacen.iVisionSensorAlmacen > 0  THEN
				i:= 0;
				bAlmacenGuardando := TRUE;
				LECTURA := DINT_TO_COLOR(ENTRADA:= GVL_Almacen.iVisionSensorAlmacen);
				GVL_Almacen.bLoadingConveyor := TRUE;
			END_IF
			
			IF fTrigRRefSensorAlmacen.Q THEN
				bAlmacenOcupado := TRUE;
				GVL_Almacen.bLoadingConveyor := FALSE;
				GVL_Almacen.sStackCraneRack.Lift:= TRUE;
			END_IF
			
			IF fTrigLift.Q THEN
				GVL_Almacen.sStackCraneRack.Right := FALSE;
			END_IF
			
			IF GVL_Almacen.sStackCraneRack.MiddleLimit THEN
				ALMACEN := CALMACEN_BUSQUEDA;
			END_IF
	END_IF
	
	CALMACEN_BUSQUEDA:
	(* Una vez colocada la caja en posición, buscamos un sitio donde almacenar *)
	
		FOR i := 1 TO 54 BY 1 DO
			IF	GVL_Almacen.aAlmacen[i] = VACIO THEN
				iPosicion := i;
				GVL_Almacen.aAlmacen[i] := LECTURA;
				ALMACEN := CALMACEN_GUARDADO;
				EXIT;
			END_IF
	
		END_FOR
	
		IF i = 55 THEN
			bEstoyLleno := TRUE;
			ALMACEN := CALMACEN_LLENO;
		END_IF
	
	
	CALMACEN_GUARDADO:
	(* Almacenamos en el sitio indicado *)
	
		GVL_Almacen.sStackCraneRack.TargetPosition := iPosicion;
		
		IF fTrigMovingX.Q THEN
			GVL_Almacen.sStackCraneRack.Left := TRUE;
		END_IF
		
		IF GVL_Almacen.sStackCraneRack.LeftLimit THEN
			GVL_Almacen.sStackCraneRack.Lift := FALSE;
			ALMACEN := CALMACEN_ORIGEN;
		END_IF	
	
	
	CALMACEN_ORIGEN:
	(* Devolvemos el almacén a posición de origen *)
	
		IF fTrigLift.Q THEN
			GVL_Almacen.sStackCraneRack.Left := FALSE;	
			
			IF LECTURA = AZUL THEN
				iCantidadAzul  := iCantidadAzul  + 1;
			END_IF
			
			IF LECTURA = VERDE THEN
				iCantidadVerde  := iCantidadVerde  + 1;
			END_IF
			
			IF LECTURA = METAL THEN
				iCantidadMetal  := iCantidadMetal + 1;
			END_IF
			
		END_IF
		
		IF GVL_Almacen.sStackCraneRack.MiddleLimit THEN
			ALMACEN := CALMACEN_ESPERA;
		END_IF
	
	
	CALMACEN_LLENO:
	(* Almacen lleno *)
	
		GVL_ProcesoPallet.sRollerConveyor.bRollerAlmacen2 := FALSE;
		GVL_ProcesoPallet.sRollerConveyor.bCurvedRollerAlmacen := FALSE;
		GVL_ProcesoPallet.sRollerConveyor.bRollerAlmacen1 := FALSE;
		
		IF NOT bEstoyLleno THEN
			ALMACEN := 0;
		END_IF
		
		ALMACEN := CALMACEN_BUSQUEDA;
	
END_CASE

END_PROGRAM

// ---- POUs/4_Almacen/PRG_RetiradaAlmacen.TcPOU
PROGRAM PRG_RetiradaAlmacen
VAR
	
	// Variables para almacenar la posición de almacenamiento y para el control del FOR
	iPosicion : INT;
	j: INT := 1;
	
	// Variable de control para conocer el estado de la máquina y permitir su coordinación con el proceso del almacén
	AlmacenSacando: BOOL;
	
	// VALORES DEL CASE
	SELECCION: CRETIRADA := CRETIRADA_ESPERA;
	
	// Function Blocks de cambios de flanco, timers...
	fTrigRRefSensorAlmacen	: F_TRIG;
	fTrigLift				: F_TRIG;
	rTrigLift				: F_TRIG;
	fTrigMovingX			: F_TRIG;
	tTimerRack 				: TON;
	tTimerRack2 			: TON;

END_VAR

fTrigRRefSensorAlmacen(CLK:= GVL_Almacen.bRRflexSensorAlmacen);
fTrigLift(CLK:= GVL_Almacen.sStackCraneRack.MovingZ);
rTrigLift(CLK:= GVL_Almacen.sStackCraneRack.MovingZ);
fTrigMovingX(CLK:= GVL_Almacen.sStackCraneRack.MovingX);
tTimerRack(IN:=GVL_Almacen.sStackCraneRack.Lift, PT:=T#1S);
tTimerRack2(IN:=GVL_Almacen.sStackCraneRack.Lift, PT:=T#3S);

(* Dejamos activadas las cintas durante todo el proceso *)

GVL_ProcesoPallet.sRollerConveyor.bRollerAlmacen3 := TRUE;
GVL_ProcesoPallet.sRollerConveyor.bRollerAlmacen4 := TRUE;

CASE SELECCION OF

	CRETIRADA_ESPERA:
	(* Si existe solicitud de salida del almacén y se ha terminado el proceso de guardado, se podrá activar el
	   proceso de salida del almacén, cambiando el valor del CASE *)
	
		IF PRG_PanelDeControl.iSolicitud > 0 AND NOT PRG_Almacen.bAlmacenGuardando THEN
			AlmacenSacando := TRUE;
			SELECCION := CRETIRADA_BUSQUEDA;
			j := 0;
		
		END_IF
		
	CRETIRADA_BUSQUEDA:
	(* El almacén busca la primera posición con el color solicitado a través del selector *)
	
		GVL_Almacen.sStackCraneRack.Left := FALSE;
		IF PRG_PanelDeControl.iSolicitud > 0 THEN
			FOR j := 1 TO 54 DO
				IF	GVL_Almacen.aAlmacen[j] = PRG_PanelDeControl.iSolicitudColor THEN
					iPosicion := j;
					GVL_Almacen.aAlmacen[j] := VACIO;
					SELECCION := CRETIRADA_RECOGIDA;
					EXIT;
				ELSIF j = 55 THEN
					SELECCION := CRETIRADA_ESPERA;
				END_IF
			END_FOR
		ELSE
			SELECCION := 1;
		END_IF
	
	CRETIRADA_RECOGIDA:
	(* El almacén recoge la caja de la posición marcada *)

		GVL_Almacen.sStackCraneRack.Right := FALSE;
		GVL_Almacen.sStackCraneRack.Lift := FALSE;
		
		IF GVL_Almacen.sStackCraneRack.MiddleLimit THEN
			GVL_Almacen.sStackCraneRack.TargetPosition := iPosicion;
		END_IF
		
		IF fTrigMovingX.Q THEN
			GVL_Almacen.sStackCraneRack.Left := TRUE;
		END_IF
		
		IF GVL_Almacen.sStackCraneRack.LeftLimit THEN
			GVL_Almacen.sStackCraneRack.Lift := TRUE;
			SELECCION := CRETIRADA_TRANSPORTE;
		END_IF	
	
	CRETIRADA_TRANSPORTE:
	(* El almacén lleva la caja a su sitio *)
	
		IF fTrigLift.Q THEN
			GVL_Almacen.sStackCraneRack.Left := FALSE;
		END_IF
		
		IF GVL_Almacen.sStackCraneRack.MiddleLimit AND NOT GVL_Almacen.sStackCraneRack.MovingZ THEN
			GVL_Almacen.sStackCraneRack.TargetPosition := 55;
		END_IF
		
		IF fTrigMovingX.Q AND GVL_Almacen.sStackCraneRack.TargetPosition = 55 THEN
			GVL_Almacen.sStackCraneRack.Lift := TRUE;
			SELECCION := CRETIRADA_COLOCACION;
		END_IF

	CRETIRADA_COLOCACION:
	(* El almacén se coloca para depositar la caja sobre el LoadingConveyor *)
	
		IF tTimerRack2.Q THEN
			GVL_Almacen.sStackCraneRack.Left := TRUE;
			SELECCION := CRETIRADA_PARTIDA;
		END_IF	
	
	CRETIRADA_PARTIDA:
	(* Una vez colocado, desciende hasta dejar la caja sobre los rodillos y dejarla partir *)

		IF GVL_Almacen.sStackCraneRack.LeftLimit THEN
			GVL_Almacen.sStackCraneRack.Lift := FALSE;
			
			IF fTrigLift.Q THEN
				
				IF PRG_PanelDeControl.iSolicitudColor = AZUL THEN
					PRG_Almacen.iCantidadAzul := PRG_Almacen.iCantidadAzul - 1;
				END_IF
				
				IF PRG_PanelDeControl.iSolicitudColor = VERDE THEN
					PRG_Almacen.iCantidadVerde := PRG_Almacen.iCantidadVerde - 1;
				END_IF
				
				IF PRG_PanelDeControl.iSolicitudColor = METAL THEN
					PRG_Almacen.iCantidadMetal := PRG_Almacen.iCantidadMetal - 1;
				END_IF
				
				PRG_PanelDeControl.iSolicitud := PRG_PanelDeControl.iSolicitud - 1;
				AlmacenSacando := FALSE;
				SELECCION := CRETIRADA_BUSQUEDA;
				
			END_IF
		END_IF
		
END_CASE

END_PROGRAM

// ---- POUs/4_Almacen/PRG_PanelDeControl.TcPOU
PROGRAM PRG_PanelDeControl
VAR
	
	// FB de cambio de flanco para la detección de las pulsaciones del botón verde
	tRTrigSacar			: R_TRIG;
	
	// Memoria para la pulsación del paro
	bReset : BOOL;
	
	// Memoria para determinar qué color se está seleccionando en cada momento
	iSolicitudColor: COLOR;
	
END_VAR

VAR_INPUT
	
	// Variable que almacena la cantidad de cajas que el operario desea sacar
	iSolicitud: INT := 0;
	
END_VAR

tRTrigSacar(CLK:= GVL_Almacen.Sacar);

(* Aquí sumamos el número de cajas a sacar por cada pulsación del botón verde *)

IF tRTrigSacar.Q THEN
	iSolicitud := iSolicitud + 1;
END_IF

(* BOTÓN NARANJA. Paro fin de ciclo *)

IF GVL_Almacen.bReset THEN
	bReset := TRUE;
END_IF

IF bReset AND PRG_RetiradaAlmacen.SELECCION > 2 THEN
	iSolicitud := 1;
END_IF


(* Rosca de selección del tipo de caja. Activa y desactiva los LEDs correspondientes y almacena en una memoria qué solicitud se está haciendo *)
	
IF GVL_Almacen.sSelector.StateAzul THEN
	GVL_Almacen.LedAzul := TRUE;
	GVL_Almacen.LedVerde := FALSE;
	GVL_Almacen.LedMetal := FALSE;
	iSolicitudColor := AZUL;
	GVL_Almacen.iDisplay := PRG_Almacen.iCantidadAzul;
END_IF

IF NOT GVL_Almacen.sSelector.StateMetal AND NOT GVL_Almacen.sSelector.StateAzul THEN
	GVL_Almacen.LedAzul := FALSE;
	GVL_Almacen.LedVerde := TRUE;
	GVL_Almacen.LedMetal := FALSE;
	iSolicitudColor := VERDE;
	GVL_Almacen.iDisplay := PRG_Almacen.iCantidadVerde;
END_IF

IF GVL_Almacen.sSelector.StateMetal THEN
	GVL_Almacen.LedAzul := FALSE;
	GVL_Almacen.LedVerde := FALSE;
	GVL_Almacen.LedMetal := TRUE;
	iSolicitudColor := METAL;
	GVL_Almacen.iDisplay := PRG_Almacen.iCantidadMetal;
END_IF

END_PROGRAM

// ---- POUs/4_Almacen/DINT_TO_COLOR.TcPOU
FUNCTION_BLOCK DINT_TO_COLOR
VAR_INPUT
	ENTRADA: DINT;
END_VAR
VAR_OUTPUT
	SALIDA: COLOR;
END_VAR
VAR

END_VAR

CASE ENTRADA OF
	2:
	SALIDA := AZUL;
	
	5:
	SALIDA := VERDE;
	
	8:
	SALIDA := METAL;
END_CASE

END_FUNCTION_BLOCK

// ---- POUs/0_ControlEncendido/PRG_FinDeCiclo.TcPOU
PROGRAM PRG_FinDeCiclo
VAR
	// Memorias que permiten que la fábrica se vaya apagando progresivamente
	bMemoriaP1 : BOOL;
	bMemoriaP2 : BOOL;
	bMemoriaP3 : BOOL;
	bMemoriaP4 : BOOL;
END_VAR


(* Cuando el operario pulsa fin de ciclo, se deja de ejecutar el bON de Main, saltando únicamente a este PRG que controla el apagado 
progresivo de los diferentes POUs. Para ello, comprueba el valor de las memorias colocadas por todo el proceso, unas superpuestas a las otras,
permitiendo encender y apagar cada estación en función de su estado de procesamiento *)

	
GVL_General.sBeltConveyor.bSortingCintaInicial := FALSE;
GVL_General.sBeltConveyor.bSortingCintaEntrada := FALSE;	


IF POU_Contadores.iCintaProcesando > 0 THEN
	PRG_OnFabrica();
	PRG_ProcesoEntrada();
	bMemoriaP1 := TRUE;
ELSE
	bMemoriaP1 := FALSE;
END_IF

IF POU_Contadores.iStackBoxProcesando > 0 OR bMemoriaP1 THEN
	PRG_PickAndPlace();
	PRG_Positioner();
	PRG_Parada();
	bMemoriaP2 := TRUE;
ELSE
	bMemoriaP2 := FALSE;
END_IF

IF POU_Contadores.iCajaProcesando > 0 OR bMemoriaP2 THEN	
	PRG_Turntable();
	bMemoriaP3 := TRUE;
ELSE
	bMemoriaP3 := FALSE;
END_IF
	
IF POU_Contadores.iProcesandoCintas > 0 OR bMemoriaP3 THEN
	PRG_Almacen();
	bMemoriaP4 := TRUE;
ELSE
	bMemoriaP4 := FALSE;
END_IF	

IF POU_Contadores.bGuardandoCaja OR bMemoriaP4 THEN
	PRG_Almacen();
	GVL_ProcesoPallet.sRollerConveyor.bRollerAlmacen1 := TRUE;
	GVL_ProcesoPallet.sRollerConveyor.bRollerAlmacen2 := TRUE;
	GVL_ProcesoPallet.sRollerConveyor.bCurvedRollerAlmacen := TRUE;
ELSE
	GVL_ProcesoPallet.sRollerConveyor.bRollerAlmacen1 := FALSE;
	GVL_ProcesoPallet.sRollerConveyor.bRollerAlmacen2 := FALSE;
	GVL_ProcesoPallet.sRollerConveyor.bCurvedRollerAlmacen := FALSE;
END_IF

IF POU_Contadores.iStackBoxProcesando = 0 THEN
	GVL_General.sBeltConveyor.bCintaAzul1 	:= FALSE;
	GVL_General.sBeltConveyor.bCintaVerde1	:= FALSE;
	GVL_General.sBeltConveyor.bCintaMetal1 	:= FALSE;
	GVL_General.sBeltConveyor.bCintaAzul2 	:= FALSE;
	GVL_General.sBeltConveyor.bCintaVerde2 	:= FALSE;
	GVL_General.sBeltConveyor.bCintaMetal2 	:= FALSE;
	GVL_General.sBeltConveyor.bSortingCintaDistribucion := FALSE;
ELSE
	GVL_General.sBeltConveyor.bCintaAzul1 	:= TRUE;
	GVL_General.sBeltConveyor.bCintaVerde1	:= TRUE;
	GVL_General.sBeltConveyor.bCintaMetal1 	:= TRUE;
	GVL_General.sBeltConveyor.bCintaAzul2 	:= TRUE;
	GVL_General.sBeltConveyor.bCintaVerde2 	:= TRUE;
	GVL_General.sBeltConveyor.bCintaMetal2 	:= TRUE;
	GVL_General.sBeltConveyor.bSortingCintaDistribucion := TRUE;
END_IF

END_PROGRAM

// ---- POUs/0_ControlEncendido/PRG_OnFabrica.TcPOU
PROGRAM PRG_OnFabrica
VAR
END_VAR

(* Este PRG activa las cintas de la fábrica necesarias para el funcionamiento inicial, y cuyo valor no variará a lo largo del proceso *)

GVL_General.sBeltConveyor.bSortingCintaInicial := TRUE;
GVL_General.sBeltConveyor.bSortingCintaEntrada := TRUE;
GVL_General.sBeltConveyor.bSortingCintaDistribucion := TRUE;

GVL_General.sBeltConveyor.bCintaAzul2 := TRUE;
GVL_General.sBeltConveyor.bCintaVerde2 := TRUE;
GVL_General.sBeltConveyor.bCintaMetal2 := TRUE;

GVL_ProcesoPallet.sRollerConveyor.bRollerAlmacen1 := TRUE;
GVL_ProcesoPallet.sRollerConveyor.bCurvedRollerAlmacen := TRUE;

END_PROGRAM

// ---- POUs/1_ProcesoEntrada/PRG_ProcesoEntrada.TcPOU
PROGRAM PRG_ProcesoEntrada
VAR
	PusherAzul: FB_Pusher;
	PusherVerde: FB_Pusher;
	PusherMetal: FB_Pusher;
END_VAR

(*Este POU se encarga de controlar la parte inicial del proceso, donde se separan los materiales de 
entrada por tipo. Para ello, se activa el proceso con el botón principal (botón MARCHA) y comienzan 
a moverse las diferentes cintas, activando los pushers cuando la detección corresponda con el objeto 
deseado. Si el sensor visual detecta el objeto configurado en sus características, entonces se pasa 
a detectar el flanco de bajada del Diffuse Sensor, activando los pushers en el momento adecuado *)

// SECCIÓN AZUL
PusherAzul(
	SENSOR:= GVL_Sorting.bDiffuseSensorA, FRONTAL:= GVL_Sorting.sPusherA.PusherFrontLimit, 
	CAMARA:= GVL_Sorting.bVisionSensorA, BLOQUEOPUSHER := PRG_Parada.bBloqueoPusherA, PUSHER=> GVL_Sorting.sPusherA.Pusher);

// SECCIÓN VERDE
PusherVerde(
	SENSOR:= GVL_Sorting.bDiffuseSensorV, FRONTAL:= GVL_Sorting.sPusherV.PusherFrontLimit, 
	CAMARA:= GVL_Sorting.bVisionSensorV, BLOQUEOPUSHER := PRG_Parada.bBloqueoPusherV, PUSHER=> GVL_Sorting.sPusherV.Pusher);

// SECCIÓN METAL
PusherMetal(
	SENSOR:= GVL_Sorting.bDiffuseSensorM, FRONTAL:= GVL_Sorting.sPusherM.PusherFrontLimit, 
	CAMARA:= GVL_Sorting.bVisionSensorM, BLOQUEOPUSHER := PRG_Parada.bBloqueoPusherM, PUSHER=> GVL_Sorting.sPusherM.Pusher);

END_PROGRAM

// ---- POUs/1_ProcesoEntrada/FB_Pusher.TcPOU
FUNCTION_BLOCK FB_Pusher
VAR_INPUT
	SENSOR : BOOL;
	FRONTAL	: BOOL;
	CAMARA : BOOL;
	BLOQUEOPUSHER : BOOL;
END_VAR
VAR_OUTPUT
	PUSHER : BOOL;
END_VAR
VAR
	FTRIGA : F_TRIG;
END_VAR

FTRIGA(CLK:= SENSOR);

IF CAMARA AND FTRIGA.Q AND NOT BLOQUEOPUSHER THEN
	PUSHER := TRUE;	 
END_IF

IF FRONTAL THEN
	PUSHER := FALSE;
END_IF

END_FUNCTION_BLOCK

// ---- POUs/2_ProcesoGuardado/PRG_Parada.TcPOU
PROGRAM PRG_Parada
VAR
	EstoyBloqueandoA: BOOL;
	EstoyBloqueandoV: BOOL;
	EstoyBloqueandoM: BOOL;

	StopBladeA: FB_StopBlade;
	CintaA: 	FB_Cinta;
	
	StopBladeV: FB_StopBlade;
	CintaV: 	FB_Cinta;
	
	StopBladeM: FB_StopBlade;
	CintaM: 	FB_Cinta;
	
	bBloqueoPusherA: BOOL;
	bBloqueoPusherV: BOOL;
	bBloqueoPusherM: BOOL;
END_VAR

(* Mediante este POU se controla el apagado de las líneas en caso de que comiencen a entrar demasiadas piezas en una misma
línea. Mediante su llamada, se impide que haya más de 3 piezas siendo procesadas simultáneamente por cada una de las líneas
del proceso de guardado en cajas. La detención se realiza mediante una llamada a los stopblades que impiden la entrada de
nuevas piezas a los positioner y, a su vez, detiene la cinta de entrada a cada una de las líneas del proceso, impidiendo que
se junten dos piezas seguidas, lo que ocasionaría el colapso total de la línea. *)

// SECCIÓN AZUL
StopBladeA(
	TENERPIEZA:= PRG_Positioner.TengoUnaPiezaA, ESTOYBLOQUEANDO=> EstoyBloqueandoA, 
	STOPBLADE=>GVL_StackBox.bStopBladeA1 );
	
CintaA(
	BLOQUEANDO:= EstoyBloqueandoA, SENSOR:= GVL_StackBox.bRReflectiveSensorA2, 
	CINTA=> GVL_General.sBeltConveyor.bCintaAzul1);

// SECCIÓN VERDE
StopBladeV(
	TENERPIEZA:= PRG_Positioner.TengoUnaPiezaV, ESTOYBLOQUEANDO=> EstoyBloqueandoV, 
	STOPBLADE=>GVL_StackBox.bStopBladeV1 );

CintaV(
	BLOQUEANDO:= EstoyBloqueandoV, SENSOR:= GVL_StackBox.bRReflectiveSensorV2, 
	CINTA=> GVL_General.sBeltConveyor.bCintaVerde1);

// SECCIÓN METAL
StopBladeM(
	TENERPIEZA:= PRG_Positioner.TengoUnaPiezaM, ESTOYBLOQUEANDO=> EstoyBloqueandoM, 
	STOPBLADE=>GVL_StackBox.bStopBladeM1 );

CintaM(
	BLOQUEANDO:= EstoyBloqueandoM, SENSOR:= GVL_StackBox.bRReflectiveSensorM2, 
	CINTA=> GVL_General.sBeltConveyor.bCintaMetal1);


// CONTROL DE ENTRADA	

(* Se tiene en cuenta el llenado de una línea. En caso de que una línea no pueda continuar abarcando
la entrada de piezas, se impide la activación del pusher correspondiente. (Se puede hacer en un FB, no
está hecho así porque me estoy muriendo *)

IF (
	PRG_Positioner.TengoUnaPiezaA AND PRG_PickAndPlace.RobotSeMueveA 
		AND EstoyBloqueandoA AND NOT GVL_General.sBeltConveyor.bCintaAzul1 ) 
THEN
	bBloqueoPusherA := TRUE;
ELSE
	bBloqueoPusherA := FALSE;
END_IF

IF (
	PRG_Positioner.TengoUnaPiezaV AND PRG_PickAndPlace.RobotSeMueveV 
		AND EstoyBloqueandoV AND NOT GVL_General.sBeltConveyor.bCintaVerde1 ) 
THEN
	bBloqueoPusherV := TRUE;
ELSE
	bBloqueoPusherV := FALSE;
END_IF	

IF (
	PRG_Positioner.TengoUnaPiezaM AND PRG_PickAndPlace.RobotSeMueveM 
		AND EstoyBloqueandoM AND NOT GVL_General.sBeltConveyor.bCintaMetal1) 
THEN
	bBloqueoPusherM := TRUE;
ELSE
	bBloqueoPusherM := FALSE;
END_IF

END_PROGRAM

// ---- POUs/2_ProcesoGuardado/FB_StopBlade.TcPOU
FUNCTION_BLOCK FB_StopBlade
VAR_INPUT
	TENERPIEZA: BOOL;
END_VAR
VAR_OUTPUT
	ESTOYBLOQUEANDO: BOOL;
	STOPBLADE: BOOL;
END_VAR
VAR
	CSTOPBLADE: STOPBLADE := STOPBLADE_REPOSO;

END_VAR

(* El StopBlade está en estado de reposo hasta recibir instrucciones *)
IF TENERPIEZA THEN
		STOPBLADE := TENERPIEZA;
		ESTOYBLOQUEANDO:= TENERPIEZA;
ELSE
		STOPBLADE := TENERPIEZA;
		ESTOYBLOQUEANDO:= TENERPIEZA;
END_IF

END_FUNCTION_BLOCK

// ---- POUs/2_ProcesoGuardado/FB_Cinta.TcPOU
FUNCTION_BLOCK FB_Cinta
VAR_INPUT
	BLOQUEANDO: BOOL;
	SENSOR: BOOL;
END_VAR
VAR_OUTPUT
	CINTA: BOOL;
END_VAR
VAR
	CCINTA: CINTA;
END_VAR

CASE CCINTA OF
	CINTA_ACTIVADO: 
	(* La cinta está trabajando normalmente a la espera de instrucciones *)
	CINTA := TRUE;
	IF BLOQUEANDO AND NOT SENSOR THEN
		CCINTA := CINTA_REPOSO;
	END_IF
	
	CINTA_REPOSO:
	(* La cinta se debe detener por la acción del sensor (pieza en espera) *)
	CINTA := FALSE;
	IF NOT BLOQUEANDO THEN
		CCINTA := CINTA_ACTIVADO;
	END_IF
END_CASE

END_FUNCTION_BLOCK

// ---- POUs/2_ProcesoGuardado/PRG_Positioner.TcPOU
PROGRAM PRG_Positioner
VAR
(* =============================================================================================== *)
(*                                  CONTROL DE LOS POSITIONER                                      *)
(* =============================================================================================== *)
(* ---------------------------------------- PIEZAS AZULES ---------------------------------------- *)
	PositionerA: FB_Positioner;
	TengoUnaPiezaA : BOOL;
	
(* ---------------------------------------- PIEZAS VERDES ---------------------------------------- *)

	PositionerV: FB_Positioner;
	TengoUnaPiezaV : BOOL;
	
(* ---------------------------------------- PIEZAS METAL ----------------------------------------- *)
	PositionerM: FB_Positioner;
	TengoUnaPiezaM : BOOL;
END_VAR

(* El Positioner se encarga de centrar las piezas. Para ello, se tiene que controlar su activación en
función de la velocidad de procesado de la estación siguiente (el Pick-And-Place. Para ello, se agregan
variables que permiten conocer el estado del robot siguiente, apagando o encendiendo los procesos del
Positioner en funciión de sus tiempos de procesado. Además, se ajusta mediante timers la velocidad de 
bajada del positioner, permitiendo que las piezas pasen correctamente por la línea *)

// PIEZAS AZULES
PositionerA(
	SENSOR1:= GVL_StackBox.bRReflectiveSensorA1, SENSOR3:= GVL_StackBox.bRReflectiveSensorA3, 
	SENSORPYP:= GVL_StackBox.bDiffuseSensorPyPA, CLAMPED:= GVL_StackBox.sPosLeftBarA.bClamped, 
	ROBOTSEMUEVE:= PRG_PickAndPlace.RobotSeMueveA, LIMITE:= GVL_StackBox.sPosLeftBarA.bLimit, 
	TENGOUNAPIEZA=> TengoUnaPiezaA, RAISE=> GVL_StackBox.sPosLeftBarA.bRaise, 
	CLAMP=> GVL_StackBox.sPosLeftBarA.bClamp );

// PIEZAS VERDES
PositionerV(
	SENSOR1:= GVL_StackBox.bRReflectiveSensorV1, SENSOR3:= GVL_StackBox.bRReflectiveSensorV3, 
	SENSORPYP:= GVL_StackBox.bDiffuseSensorPyPV, CLAMPED:= GVL_StackBox.sPosLeftBarV.bClamped, 
	ROBOTSEMUEVE:= PRG_PickAndPlace.RobotSeMueveV, LIMITE:= GVL_StackBox.sPosLeftBarV.bLimit, 
	TENGOUNAPIEZA=> TengoUnaPiezaV, RAISE=> GVL_StackBox.sPosLeftBarV.bRaise, 
	CLAMP=> GVL_StackBox.sPosLeftBarV.bClamp );

// PIEZAS METAL
PositionerM(
	SENSOR1:= GVL_StackBox.bRReflectiveSensorM1, SENSOR3:= GVL_StackBox.bRReflectiveSensorM3, 
	SENSORPYP:= GVL_StackBox.bDiffuseSensorPyPM, CLAMPED:= GVL_StackBox.sPosLeftBarM.bClamped, 
	ROBOTSEMUEVE:= PRG_PickAndPlace.RobotSeMueveM, LIMITE:= GVL_StackBox.sPosLeftBarM.bLimit, 
	TENGOUNAPIEZA=> TengoUnaPiezaM, RAISE=> GVL_StackBox.sPosLeftBarM.bRaise, 
	CLAMP=> GVL_StackBox.sPosLeftBarM.bClamp );

END_PROGRAM

// ---- POUs/2_ProcesoGuardado/FB_Positioner.TcPOU
FUNCTION_BLOCK FB_Positioner
VAR_INPUT
	
	SENSOR1 : BOOL;
	SENSOR3 : BOOL;
	SENSORPYP : BOOL;
	CLAMPED : BOOL;
	ROBOTSEMUEVE : BOOL;
	LIMITE : BOOL;
	
END_VAR
VAR_OUTPUT
	
	TENGOUNAPIEZA : BOOL := FALSE;
	CLAMP : BOOL;
	RAISE : BOOL;
	
END_VAR
VAR
	CPOSITIONERLEFTBAR		 : CPOSITIONERLEFTBAR := CPOSITIONERLEFTBAR_ESPERA;

	tClampTimer				 : TON;
	tClampTimer2			 : TON;
	
	bRTrigClamp				 : R_TRIG;	
	bRTrigRReflectiveSensor1 : R_TRIG;
	bFTrigDifSensorPyP		 : F_TRIG;
	bRTrigRReflectiveSensor3 : R_TRIG;

END_VAR

bRTrigClamp(CLK:= RAISE);
tClampTimer(IN:= RAISE, PT:= T#0.7S);

bRTrigRReflectiveSensor1(CLK:= SENSOR1);
bRTrigRReflectiveSensor3(CLK:= SENSOR3);
bFTrigDifSensorPyP(CLK:= SENSORPYP);

(* Se fuerza que el positioner solo funcione cuando el sensor inmediatamente anterior, detecta un cambio
de flanco. Para evitar el golpe inicial de inicio de fábrica, se le añade el control a través del botón de
marcha, aprovechando que se mantiene un pequeño período de tiempo pulsado *)

IF bRTrigRReflectiveSensor3.Q AND NOT GVL_General.bMarcha THEN
	TENGOUNAPIEZA := TRUE;
END_IF

(* Se definen los CASE para su control. Se definen etapas correspondientes a los diferentes estados
en los que se debe encontrar para su funcionamiento. Además, se controla el número de elementos
simultáneos en la cinta a través de la variable iContadorCX2 (siendo X el tipo de línea) *)
	
CASE CPOSITIONERLEFTBAR OF
	
	CPOSITIONERLEFTBAR_ESPERA:
	(* Aqui la maquina esta esperando a que sea su turno para funcionar *)	
	
		IF TENGOUNAPIEZA THEN
			CPOSITIONERLEFTBAR := CPOSITIONERLEFTBAR_AGARRE;
		END_IF

	CPOSITIONERLEFTBAR_AGARRE:
	(* El proceso activa mediante el cambio de flanco del sensor el agarre del objeto de 
	entrada. Se añade una variable bOn que mantiene el sistema encendido hasta el siguiente cambio 
	de flanco, controlando correctamente la barrera de entrada *)
	
		CLAMP := TRUE;
		
		IF CLAMPED  AND NOT ROBOTSEMUEVE THEN
			CPOSITIONERLEFTBAR := CPOSITIONERLEFTBAR_PROCESADO;
		END_IF		
	
	CPOSITIONERLEFTBAR_PROCESADO:
	(* El objeto se suelta una vez colocado correctamente en la cinta, y se eleva el Positioner para
	permitir su avance por la línea. *)
	
		CLAMP := FALSE;
		RAISE := TRUE;
		
		IF bRTrigClamp.Q THEN 
			CPOSITIONERLEFTBAR := CPOSITIONERLEFTBAR_RESET;
		END_IF
	
	CPOSITIONERLEFTBAR_RESET:
	(* Se baja el Positioner hasta que vuelve a su posición inicial. Se agrega un timer que permite
	esperar a que el LID correspondiente se encuentre fuera del rango de la máquina, para evitar 
	colisiones sobre el material. Una vez esto ocurre, se abre el paso para el siguiente elemento *)

		IF LIMITE AND tClampTimer.Q THEN
			RAISE := FALSE;
			CPOSITIONERLEFTBAR := CPOSITIONERLEFTBAR_PASO;
		END_IF	
	
	CPOSITIONERLEFTBAR_PASO: 
	(* La barrera no se bajará hasta qe el positioner llegue al final de su movimiento *)
	
		IF LIMITE THEN
			TENGOUNAPIEZA := FALSE;
			CPOSITIONERLEFTBAR := CPOSITIONERLEFTBAR_ESPERA;
		END_IF
END_CASE

END_FUNCTION_BLOCK

// ---- POUs/3_ProcesoPalet/PRG_Cintas.TcPOU
PROGRAM PRG_Cintas
VAR
END_VAR


(* Dependiendo de las detecciones de los sensores, se activarán según qué líneas*)

IF NOT PRG_PickAndPlace.CajaLlenaA THEN
	IF GVL_ProcesoPallet.iLightArrayEmitterA THEN
		GVL_ProcesoPallet.sRollerConveyor.bRollerAzul1 := FALSE;
	ELSE
		GVL_ProcesoPallet.sRollerConveyor.bRollerAzul1 := TRUE;
	END_IF
END_IF

IF NOT PRG_PickAndPlace.CajaLlenaV THEN
	IF GVL_ProcesoPallet.iLightArrayEmitterV THEN
		GVL_ProcesoPallet.sRollerConveyor.bRollerVerde1 := FALSE;
	ELSE
		GVL_ProcesoPallet.sRollerConveyor.bRollerVerde1 := TRUE;
	END_IF
END_IF

IF NOT PRG_PickAndPlace.CajaLlenaM THEN
	IF GVL_ProcesoPallet.iLightArrayEmitterM THEN
		GVL_ProcesoPallet.sRollerConveyor.bRollerMetal1 := FALSE;
	ELSE
		GVL_ProcesoPallet.sRollerConveyor.bRollerMetal1 := TRUE;
	END_IF
END_IF

END_PROGRAM

// ---- POUs/0_ControlEncendido/PRG_SetaEmergencia.TcPOU
PROGRAM PRG_SetaEmergencia
VAR
END_VAR

(* GVL GENERAL *)

GVL_General.sBeltConveyor.bSortingCintaDistribucion := FALSE;
GVL_General.sBeltConveyor.bSortingCintaEntrada := FALSE;
GVL_General.sBeltConveyor.bSortingCintaInicial := FALSE;


GVL_General.bStopBlade1 := FALSE;


GVL_General.sBeltConveyor.bCintaAzul1 := FALSE;
GVL_General.sBeltConveyor.bCintaAzul2 := FALSE;

GVL_General.sBeltConveyor.bCintaMetal1 := FALSE;
GVL_General.sBeltConveyor.bCintaMetal2 := FALSE;

GVL_General.sBeltConveyor.bCintaVerde1 := FALSE;
GVL_General.sBeltConveyor.bCintaVerde2 := FALSE;


(* GVL SORTING *)

GVL_Sorting.sPusherA.Pusher := FALSE;
GVL_Sorting.sPusherV.Pusher := FALSE;
GVL_Sorting.sPusherM.Pusher := FALSE;


(* GVL STACKBOX *)

GVL_StackBox.bStopBladeA1 := FALSE;
GVL_StackBox.bStopBladeA2 := FALSE;

GVL_StackBox.bStopBladeV1 := FALSE;
GVL_StackBox.bStopBladeV2 := FALSE;

GVL_StackBox.bStopBladeM1 := FALSE;
GVL_StackBox.bStopBladeM2 := FALSE;

GVL_StackBox.sPickAndPlaceA.bGrab := FALSE;
GVL_StackBox.sPickAndPlaceA.bGripperCCW := FALSE;
GVL_StackBox.sPickAndPlaceA.bGripperCW := FALSE;
GVL_StackBox.sPickAndPlaceA.bMovementX := FALSE;
GVL_StackBox.sPickAndPlaceA.bMovementZ := FALSE;
GVL_StackBox.sPickAndPlaceA.bRotateCCW := FALSE;
GVL_StackBox.sPickAndPlaceA.bRotateCW := FALSE;

(* GVL PROCESOPALLET*)

GVL_ProcesoPallet.sTurnTable.RollNegativo := FALSE;
GVL_ProcesoPallet.sTurnTable.RollPositivo := FALSE;
GVL_ProcesoPallet.sTurnTable.Turn := FALSE;
GVL_ProcesoPallet.sRollerConveyor.bCurvedRollerAlmacen:= FALSE;
GVL_ProcesoPallet.sRollerConveyor.bCurvedRollerAzul1 := FALSE;
GVL_ProcesoPallet.sRollerConveyor.bCurvedRollerMetal1 := FALSE;
GVL_ProcesoPallet.sRollerConveyor.bRollerAlmacen1 := FALSE;
GVL_ProcesoPallet.sRollerConveyor.bRollerAlmacen2 := FALSE;
GVL_ProcesoPallet.sRollerConveyor.bRollerAlmacen3 := FALSE;
GVL_ProcesoPallet.sRollerConveyor.bRollerAlmacen4 := FALSE;
GVL_ProcesoPallet.sRollerConveyor.bRollerAzul1 := FALSE;
GVL_ProcesoPallet.sRollerConveyor.bRollerVerde1 := FALSE;
GVL_ProcesoPallet.sRollerConveyor.bRollerMetal1 := FALSE;


(*GVL ALMACEN *)

GVL_Almacen.bLoadingConveyor := FALSE;
GVL_Almacen.sStackCraneRack.Left := FALSE;
GVL_Almacen.sStackCraneRack.Lift := FALSE;
GVL_Almacen.sStackCraneRack.Right := FALSE;

END_PROGRAM
